(* IEC 61131-3 sources: exOS-Samples/WaterTank/JavaScript/Binary/WaterTank/WaterTank_0, 1 file *)

(* ---- WaterTank.st ---- *)
PROGRAM _INIT

    WaterTankInit_0();

END_PROGRAM

PROGRAM _CYCLIC

    //Auto connect:
    //WaterTankCyclic_0.Enable := ExComponentInfo_0.Operational;
    WaterTankCyclic_0(Handle := WaterTankInit_0.Handle, pWaterTank := ADR(WaterTank_0));

    ExComponentInfo_0(ExTargetLink := ADR(gTarget_0), ExComponentLink := ADR(gWaterTank_0), Enable := TRUE);

	ExDatamodelInfo_0(ExTargetLink := ADR(gTarget_0), Enable := TRUE, InstanceName := 'WaterTank_0');

	ExDataConnectionInfo_0(ExTargetLink := ADR(gTarget_0), Enable := TRUE);

END_PROGRAM

PROGRAM _EXIT

    WaterTankExit_0(Handle := WaterTankInit_0.Handle);

END_PROGRAM
